// TwinCAT 3 PLC project Sample_Delivery
// ProgramVersion: 3.1.4023.0
// libraries:
//   LCLS General, * (SLAC)
//   LCLS Vacuum, * (SLAC - LCLS)
//   Tc2_Standard, * (Beckhoff Automation GmbH)
//   Tc2_System, * (Beckhoff Automation GmbH)
//   Tc3_Module, * (Beckhoff Automation GmbH)
// project tree:
//   GVLs/ GVL_RCC.TcGVL
//   / PlcTask.TcTTO
//   POUs/ MAIN.TcPOU
// real-time tasks:
//   TASK PlcTask: cycle T#10ms, priority 20, ADS port 350
// I/O:
//   DEVICE Device 1 (EtherCAT), AmsNetId 172.21.148.84.2.1
//     Term 4 (EK1200) [EK1200-5000 EtherCAT Power supply (2A E-Bus)]
//       RCC_E1 (EL2004) [EL2004 4Ch. Dig. Output 24V, 0.5A]
//       RCC_E2 (EL1004) [EL1004 4Ch. Dig. Input 24V, 3ms]
//       RCC_E3 (EL1004) [EL1004 4Ch. Dig. Input 24V, 3ms]
//       RCC_TC (EL3314) [EL3314 4Ch. Ana. Input Thermocouple (TC)]
//       Term 9 (EK1110) [EK1110 EtherCAT extension]

CONFIGURATION Sample_Delivery
    RESOURCE PLC ON TwinCAT3
        TASK PlcTask(INTERVAL := T#10ms, PRIORITY := 20);
        PROGRAM MAIN WITH PlcTask : MAIN;
    END_RESOURCE
END_CONFIGURATION

// ---- GVLs/GVL_RCC.TcGVL
VAR_GLOBAL
    (* OverrideMode *)
    {attribute 'pytmc' := 'pv: CRIXS:RCC:VAC:OVRD_MODE'}
    xSystemOverrideMode_RCC	: BOOL := FALSE;

    (* Roughing Manifold Valvese *)

    {attribute 'pytmc' :=' pv: CRIXS:RCC:VRC:01 '}
    {attribute 'TcLinkTo' := 	'.i_xClsLS	:=	TIID^Device 1 (EtherCAT)^Term 1 (EK1200)^Term 2 (EK1122)^Hoffman Box Vac EK1 (EK1100)^VLS_RCC (EK1122)^RCC_EK0 (EK1100)^RCC_E1 (EL1004)^Channel 1^Input;
                                .q_xOPN_DO	:=	TIID^Device 1 (EtherCAT)^Term 1 (EK1200)^Term 2 (EK1122)^Hoffman Box Vac EK1 (EK1100)^VLS_RCC (EK1122)^RCC_EK0 (EK1100)^RCC_E2 (EL2004)^Channel 1^Output'}
    RCC_VRC_01 : FB_VRC_NC_ClsLS;

    (* Roughing Manifold Valvese *)

    {attribute 'pytmc' :=' pv: CRIXS:RCC:VRC:02 '}
    {attribute 'TcLinkTo' := 	'.i_xOpnLS	:=	TIID^Device 1 (EtherCAT)^Term 1 (EK1200)^Term 2 (EK1122)^Hoffman Box Vac EK1 (EK1100)^VLS_RCC (EK1122)^RCC_EK0 (EK1100)^RCC_E1 (EL1004)^Channel 4^Input;
                                 .i_xClsLS	:=	TIID^Device 1 (EtherCAT)^Term 1 (EK1200)^Term 2 (EK1122)^Hoffman Box Vac EK1 (EK1100)^VLS_RCC (EK1122)^RCC_EK0 (EK1100)^RCC_E1 (EL1004)^Channel 2^Input;
                                .q_xOPN_DO	:=	TIID^Device 1 (EtherCAT)^Term 1 (EK1200)^Term 2 (EK1122)^Hoffman Box Vac EK1 (EK1100)^VLS_RCC (EK1122)^RCC_EK0 (EK1100)^RCC_E2 (EL2004)^Channel 2^Output'}
    RCC_VRC_02 : FB_VRC;

    (* Roughing Manifold Valvese *)

    {attribute 'pytmc' :=' pv: CRIXS:RCC:VRC:03 '}
    {attribute 'TcLinkTo' := 	'.i_xClsLS	:=	TIID^Device 1 (EtherCAT)^Term 1 (EK1200)^Term 2 (EK1122)^Hoffman Box Vac EK1 (EK1100)^VLS_RCC (EK1122)^RCC_EK0 (EK1100)^RCC_E1 (EL1004)^Channel 3^Input;
                                .q_xOPN_DO	:=	TIID^Device 1 (EtherCAT)^Term 1 (EK1200)^Term 2 (EK1122)^Hoffman Box Vac EK1 (EK1100)^VLS_RCC (EK1122)^RCC_EK0 (EK1100)^RCC_E2 (EL2004)^Channel 3^Output'}
    RCC_VRC_03 : FB_VRC_NC_ClsLS;

    (* Roughing Manifold Valvese *)

    {attribute 'pytmc' :=' pv: CRIXS:RCC:VRC:04 '}
    {attribute 'TcLinkTo' := 	'.i_xClsLS	:=	TIID^Device 1 (EtherCAT)^Term 1 (EK1200)^Term 2 (EK1122)^Hoffman Box Vac EK1 (EK1100)^VLS_RCC (EK1122)^RCC_EK0 (EK1100)^RCC_E3 (EL1004)^Channel 1^Input;
                                .q_xOPN_DO	:=	TIID^Device 1 (EtherCAT)^Term 1 (EK1200)^Term 2 (EK1122)^Hoffman Box Vac EK1 (EK1100)^VLS_RCC (EK1122)^RCC_EK0 (EK1100)^RCC_E2 (EL2004)^Channel 4^Output'}
    RCC_VRC_04 : FB_VRC_NC_ClsLS;


    {attribute 'pytmc' :=' pv: CRIXS:RCC:GCP:01 '}
    {attribute 'TcLinkTo' := 	'.xPress_OK	:=	TIID^Device 1 (EtherCAT)^Term 1 (EK1200)^Term 2 (EK1122)^Hoffman Box Vac EK1 (EK1100)^VLS_RCC (EK1122)^RCC_GPI (901P)^TXPDO Combined^Combination Gauge Reading Valid;
                                 .xOverrange	:=	TIID^Device 1 (EtherCAT)^Term 1 (EK1200)^Term 2 (EK1122)^Hoffman Box Vac EK1 (EK1100)^VLS_RCC (EK1122)^RCC_GPI (901P)^TXPDO Combined^Combination Gauge Overrange Exceeded;
                                .xUnderrange := TIID^Device 1 (EtherCAT)^Term 1 (EK1200)^Term 2 (EK1122)^Hoffman Box Vac EK1 (EK1100)^VLS_RCC (EK1122)^RCC_GPI (901P)^TXPDO Combined^Combination Gauge Underrange Exceeded;
                                .i_iPRESS_R := TIID^Device 1 (EtherCAT)^Term 1 (EK1200)^Term 2 (EK1122)^Hoffman Box Vac EK1 (EK1100)^VLS_RCC (EK1122)^RCC_GPI (901P)^TXPDO Combined^Combination Gauge Active Value;
                                .bWcstate := TIID^Device 1 (EtherCAT)^Term 1 (EK1200)^Term 2 (EK1122)^Hoffman Box Vac EK1 (EK1100)^VLS_RCC (EK1122)^RCC_GPI (901P)^WcState^WcState' }
    RCC_GCP_01 : FB_901_ECAT;


    {attribute 'pytmc' :=' pv: CRIXS:RCC:01 '}
    {attribute 'TcLinkTo' := ' .bError := TIID^Device 1 (EtherCAT)^Term 1 (EK1200)^Term 2 (EK1122)^Hoffman Box Vac EK1 (EK1100)^VLS_RCC (EK1122)^RCC_EK0 (EK1100)^RCC_E7 (EL3314)^TC Inputs Channel 3^Status^Error;
                               .bUnderrange := TIID^Device 1 (EtherCAT)^Term 1 (EK1200)^Term 2 (EK1122)^Hoffman Box Vac EK1 (EK1100)^VLS_RCC (EK1122)^RCC_EK0 (EK1100)^RCC_E7 (EL3314)^TC Inputs Channel 3^Status^Underrange;
                               .bOverrange :=  TIID^Device 1 (EtherCAT)^Term 1 (EK1200)^Term 2 (EK1122)^Hoffman Box Vac EK1 (EK1100)^VLS_RCC (EK1122)^RCC_EK0 (EK1100)^RCC_E7 (EL3314)^TC Inputs Channel 3^Status^Overrange;
                               .iRaw	:= TIID^Device 1 (EtherCAT)^Term 1 (EK1200)^Term 2 (EK1122)^Hoffman Box Vac EK1 (EK1100)^VLS_RCC (EK1122)^RCC_EK0 (EK1100)^RCC_E7 (EL3314)^TC Inputs Channel 3^Value '}
   RCC_STC_01 : FB_TempSensor;
END_VAR

// ---- POUs/MAIN.TcPOU
PROGRAM MAIN
VAR
    RCC_VRC_01_OPEN_OK : BOOL;
    RCC_VRC_02_OPEN_OK : BOOL;
    RCC_VRC_03_OPEN_OK : BOOL;
    RCC_VRC_04_OPEN_OK : BOOL;

   {attribute 'pytmc' :=' pv: CRIXS:GCP:01:INLK_Setpoint '}
    RCC_GCP_01_INTERLOCK_SETPOINT : REAL := 10;
END_VAR

RCC_GCP_01(PG=>);
RCC_STC_01();

(* Valve can open only when CRIX-RCC-VRC-02 and 03 are closed*)
RCC_VRC_01_OPEN_OK := ( RCC_VRC_02.iq_stValve.i_xClsLS AND NOT RCC_VRC_02.iq_stValve.q_xOPN_DO ) AND
                                    ( RCC_VRC_03.iq_stValve.i_xClsLS AND NOT RCC_VRC_03.iq_stValve.q_xOPN_DO ) ;

RCC_VRC_01(i_xExtILK_OK := RCC_VRC_01_OPEN_OK,
                i_xOverrideMode := xSystemOverrideMode_RCC,
                 iq_stValve=> );

(* Valve can open only when CRIX-RCC-VRC-01 and 04 are closed*)
RCC_VRC_02_OPEN_OK := ( RCC_VRC_01.iq_stValve.i_xClsLS AND NOT RCC_VRC_01.iq_stValve.q_xOPN_DO ) AND
                                    ( RCC_VRC_04.iq_stValve.i_xClsLS AND NOT RCC_VRC_04.iq_stValve.q_xOPN_DO );

RCC_VRC_02(i_xExtILK_OK := RCC_VRC_02_OPEN_OK,
                i_xOverrideMode := xSystemOverrideMode_RCC,
                 iq_stValve=> );

(* Valve can open only when CRIX-RCC-GCP-01 reading < setpoint Torr and CRIX-RCC-VRC-01 and 04 are closed*)
RCC_VRC_03_OPEN_OK := (RCC_GCP_01.PG.rPRESS < RCC_GCP_01_INTERLOCK_SETPOINT and RCC_GCP_01.PG.xPRESS_OK ) AND
                                 ( RCC_VRC_01.iq_stValve.i_xClsLS AND NOT RCC_VRC_01.iq_stValve.q_xOPN_DO ) AND
                                              ( RCC_VRC_04.iq_stValve.i_xClsLS AND NOT RCC_VRC_04.iq_stValve.q_xOPN_DO );

RCC_VRC_03(i_xExtILK_OK := RCC_VRC_03_OPEN_OK,
                i_xOverrideMode := xSystemOverrideMode_RCC,
                 iq_stValve=> );

(* Valve can open only when CRIX-RCC-VRC-02 and 03 are closed*)
RCC_VRC_04_OPEN_OK := ( RCC_VRC_02.iq_stValve.i_xClsLS AND NOT RCC_VRC_02.iq_stValve.q_xOPN_DO ) AND
                                      ( RCC_VRC_03.iq_stValve.i_xClsLS AND NOT RCC_VRC_03.iq_stValve.q_xOPN_DO ) ;

RCC_VRC_04(i_xExtILK_OK := RCC_VRC_04_OPEN_OK,
                i_xOverrideMode := xSystemOverrideMode_RCC,
                 iq_stValve=> );

END_PROGRAM
